Staubli VAL3: page.pgx

public program page(string& menuname[], num index)
// set all the page in english
begin
  //
  //  PAGE
  //
    //
    // PALLET PAGE
    if index>=10 and index<=19
      title ("< Pgina Palet >")
    endIf
    // PALLET VIEW PAGE
    if index>=100 and index<=109
      title("< Visor Pgina Palet >")
    endIf
  switch index
        //
    // PALLET
    //
    // Integrator programmer
    case 10,11
      menuname="Visor Programa,Editar Palet,,,Wizard,Resetear,Atras,Siguiente"
    break
    // On Cycle
    case 13,14
      menuname="Visor Programa,Editar Palet,,,,Resetear,Atras,Siguiente"
    break
    // VIEW PALLET
    case 100,101,102,103,104,105
      menuname="Resetear TODO,,,,,Resetear,Atras,Siguiente"
    break
  endSwitch
end
